(* PLC project HomeAutomation.project, CODESYS CODESYS V3.5 SP15 Patch 1 *)
(* stored: creationDateTime 2019-10-07T17:20:35.7601886, modificationDateTime 2019-10-07T17:17:55.9764537 *)

TYPE MQTT_MESSAGE : STRUCT
  Payload : STRING(128);
  Topic : STRING(128);
  Qos : SD_MQTT.QoS;
  MqttRetain : BOOL;
END_STRUCT;
END_TYPE

TYPE COVER_STATES : (Idle, Auto, Manual, Prio_up, Prio_dn, Calibrate_up, Calibrate_dn);
END_TYPE

PROGRAM PLC_PRG_MAIN
  VAR
    MqttPushbuttonPrefix : STRING(100) := 'WAGO-PFC200/Out/DigitalInputs/Pushbuttons/';  (* INPUT FUNCTION BLOCKS *)
    FB_DI_PB_001 : FB_INPUT_PUSHBUTTON_MQTT;
    FB_DI_PB_002 : FB_INPUT_PUSHBUTTON_MQTT;
    FB_DI_PB_003 : FB_INPUT_PUSHBUTTON_MQTT;
    FB_DI_PB_004 : FB_INPUT_PUSHBUTTON_MQTT;
    FB_DI_PB_005 : FB_INPUT_PUSHBUTTON_MQTT;
    FB_DI_PB_006 : FB_INPUT_PUSHBUTTON_MQTT;
    FB_DI_PB_007 : FB_INPUT_PUSHBUTTON_MQTT;
    FB_DI_PB_008 : FB_INPUT_PUSHBUTTON_MQTT;
    FB_DI_PB_009 : FB_INPUT_PUSHBUTTON_DIMMER_MQTT;
    FB_DI_PB_010 : FB_INPUT_PUSHBUTTON_MQTT;
    FB_DI_PB_011 : FB_INPUT_PUSHBUTTON_MQTT;
    FB_DI_PB_012 : FB_INPUT_PUSHBUTTON_MQTT;
    FB_DI_PB_013 : FB_INPUT_PUSHBUTTON_MQTT;
    FB_DI_PB_014 : FB_INPUT_PUSHBUTTON_MQTT;
    FB_DI_PB_015 : FB_INPUT_PUSHBUTTON_MQTT;
    FB_DI_PB_016 : FB_INPUT_PUSHBUTTON_MQTT;
    FB_DI_PB_017 : FB_INPUT_PUSHBUTTON_MQTT;
    FB_DI_PB_018 : FB_INPUT_PUSHBUTTON_MQTT;
    FB_DI_PB_019 : FB_INPUT_PUSHBUTTON_MQTT;
    FB_DI_PB_020 : FB_INPUT_PUSHBUTTON_MQTT;
    FB_DI_PB_021 : FB_INPUT_PUSHBUTTON_MQTT;
    FB_DI_PB_022 : FB_INPUT_PUSHBUTTON_MQTT;
    FB_DI_PB_023 : FB_INPUT_PUSHBUTTON_MQTT;
    FB_DI_PB_024 : FB_INPUT_PUSHBUTTON_MQTT;
    FB_DI_PB_025 : FB_INPUT_PUSHBUTTON_MQTT;
    FB_DI_PB_026 : FB_INPUT_PUSHBUTTON_MQTT;
    FB_DI_PB_027 : FB_INPUT_PUSHBUTTON_MQTT;
    FB_DI_PB_028 : FB_INPUT_PUSHBUTTON_MQTT;
    FB_DI_PB_029 : FB_INPUT_PUSHBUTTON_MQTT;
    FB_DI_PB_030 : FB_INPUT_PUSHBUTTON_MQTT;
    FB_DI_PB_031 : FB_INPUT_PUSHBUTTON_MQTT;
    FB_DI_PB_032 : FB_INPUT_PUSHBUTTON_MQTT;
    FB_DI_PB_033 : FB_INPUT_PUSHBUTTON_MQTT;
    FB_DI_PB_034 : FB_INPUT_PUSHBUTTON_MQTT;
    FB_DI_PB_035 : FB_INPUT_PUSHBUTTON_MQTT;
    FB_DI_PB_036 : FB_INPUT_PUSHBUTTON_MQTT;
    FB_DI_PB_037 : FB_INPUT_PUSHBUTTON_MQTT;
    FB_DI_PB_038 : FB_INPUT_PUSHBUTTON_MQTT;
    FB_DI_PB_039 : FB_INPUT_PUSHBUTTON_MQTT;
    FB_DI_PB_040 : FB_INPUT_PUSHBUTTON_MQTT;
    FB_DI_PB_041 : FB_INPUT_PUSHBUTTON_MQTT;
    FB_DI_PB_042 : FB_INPUT_PUSHBUTTON_MQTT;
    FB_DI_PB_043 : FB_INPUT_PUSHBUTTON_MQTT;
    FB_DI_PB_044 : FB_INPUT_PUSHBUTTON_MQTT;
    FB_DI_PB_045 : FB_INPUT_PUSHBUTTON_MQTT;
    FB_DI_PB_046 : FB_INPUT_PUSHBUTTON_MQTT;
    FB_DI_PB_047 : FB_INPUT_PUSHBUTTON_MQTT;
    FB_DI_PB_048 : FB_INPUT_PUSHBUTTON_MQTT;
    MqttPubSwitchPrefix : STRING(100) := 'WAGO-PFC200/Out/DigitalOutputs/';  (* OUTPUT FUNCTION BLOCKS *)
    MqttSubSwitchPrefix : STRING(100) := 'WAGO-PFC200/In/DigitalOutputs/';
    FB_DO_SW_001 : FB_OUTPUT_SWITCH_MQTT;
    FB_DO_SW_002 : FB_OUTPUT_SWITCH_MQTT;
    FB_DO_SW_003 : FB_OUTPUT_SWITCH_MQTT;
    FB_DO_SW_004 : FB_OUTPUT_SWITCH_MQTT;
    FB_DO_SW_005 : FB_OUTPUT_SWITCH_MQTT;
    FB_DO_SW_006 : FB_OUTPUT_SWITCH_MQTT;
    FB_DO_SW_007 : FB_OUTPUT_SWITCH_MQTT;
    FB_DO_SW_008 : FB_OUTPUT_SWITCH_MQTT;
    FB_DO_SW_009 : FB_OUTPUT_SWITCH_MQTT;
    FB_DO_SW_010 : FB_OUTPUT_SWITCH_MQTT;
    FB_DO_SW_011 : FB_OUTPUT_SWITCH_MQTT;
    FB_DO_SW_012 : FB_OUTPUT_SWITCH_MQTT;
    FB_DO_SW_013 : FB_OUTPUT_SWITCH_MQTT;
    FB_DO_SW_014 : FB_OUTPUT_SWITCH_MQTT;
    FB_DO_SW_015 : FB_OUTPUT_SWITCH_MQTT;
    FB_DO_SW_016 : FB_OUTPUT_SWITCH_MQTT;
    FB_DO_SW_017 : FB_OUTPUT_SWITCH_MQTT;
    FB_DO_SW_018 : FB_OUTPUT_SWITCH_MQTT;
    FB_DO_SW_019 : FB_OUTPUT_SWITCH_MQTT;
    FB_DO_SW_020 : FB_OUTPUT_SWITCH_MQTT;
    FB_DO_SW_021 : FB_OUTPUT_SWITCH_MQTT;
    FB_DO_SW_022 : FB_OUTPUT_SWITCH_MQTT;
    FB_DO_SW_023 : FB_OUTPUT_SWITCH_MQTT;
    FB_DO_SW_024 : FB_OUTPUT_SWITCH_MQTT;
    FB_DO_SW_025 : FB_OUTPUT_SWITCH_MQTT;
    FB_DO_SW_026 : FB_OUTPUT_SWITCH_MQTT;
    FB_DO_SW_027 : FB_OUTPUT_SWITCH_MQTT;
    FB_DO_SW_028 : FB_OUTPUT_SWITCH_MQTT;
    FB_DO_SW_029 : FB_OUTPUT_SWITCH_MQTT;
    FB_DO_SW_030 : FB_OUTPUT_SWITCH_MQTT;
    FB_DO_SW_031 : FB_OUTPUT_SWITCH_MQTT;
    FB_DO_SW_032 : FB_OUTPUT_SWITCH_MQTT;
    MqttPubCoverPrefix : STRING(100) := 'WAGO-PFC200/Out/Covers/';  (* COVER FUNCTION BLOCKS *)
    MqttSubCoverPrefix : STRING(100) := 'WAGO-PFC200/In/Covers/';
    FB_DO_COVER_001 : FB_OUTPUT_COVER_MQTT;
  END_VAR

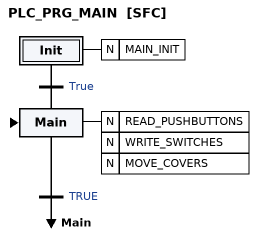
INITIAL_STEP Init:
  MAIN_INIT(N);
END_STEP
TRANSITION FROM Init TO Main
  := True;
END_TRANSITION
STEP Main:
  READ_PUSHBUTTONS(N);
  WRITE_SWITCHES(N);
  MOVE_COVERS(N);
END_STEP
TRANSITION FROM Main TO Main
  := TRUE;
END_TRANSITION

ACTION WRITE_SWITCHES:
                      FB_DO_SW_001(OUT	=>		DO_001,										(* couple the function block to the physical output *)
	PRIO_HIGH				:=FALSE,  									(* brings the output high regardless of other input values *)
	PRIO_LOW				:=FALSE, 									(* brings the output low regardless of other input values. NOTE: PRIO_HIGH overrules PRIO_LOW input *)
	TOGGLE					:=FB_DI_PB_009.SINGLE 						(* for toggling the output *)	
);

FB_DO_SW_002(OUT => DO_002		,PRIO_HIGH:=FALSE			,PRIO_LOW:=FALSE				,TOGGLE:=FB_DI_PB_009.DOUBLE	);
FB_DO_SW_003(OUT => DO_003		,PRIO_HIGH:=FALSE			,PRIO_LOW:=FALSE				,TOGGLE:=FB_DI_PB_009.LONG		);
FB_DO_SW_004(OUT => DO_004		,PRIO_HIGH:=FALSE			,PRIO_LOW:=FALSE				,TOGGLE:=FB_DI_PB_009.LONG		);
FB_DO_SW_005(OUT => DO_005		,PRIO_HIGH:=FALSE			,PRIO_LOW:=FALSE				,TOGGLE:=FB_DI_PB_009.LONG		);
FB_DO_SW_006(OUT => DO_006		,PRIO_HIGH:=FALSE			,PRIO_LOW:=FALSE				,TOGGLE:=FB_DI_PB_009.LONG		);
FB_DO_SW_007(OUT => DO_007		,PRIO_HIGH:=FALSE			,PRIO_LOW:=FALSE				,TOGGLE:=FB_DI_PB_009.LONG		);
FB_DO_SW_008(OUT => DO_008		,PRIO_HIGH:=FALSE			,PRIO_LOW:=FALSE				,TOGGLE:=FB_DI_PB_009.LONG		);
FB_DO_SW_009(OUT => DO_009		,PRIO_HIGH:=FALSE			,PRIO_LOW:=FALSE				,TOGGLE:=FALSE				);
FB_DO_SW_010(OUT => DO_010		,PRIO_HIGH:=FALSE			,PRIO_LOW:=FALSE				,TOGGLE:=FALSE				);
FB_DO_SW_011(OUT => DO_011		,PRIO_HIGH:=FALSE			,PRIO_LOW:=FALSE				,TOGGLE:=FALSE				);
FB_DO_SW_012(OUT => DO_012		,PRIO_HIGH:=FALSE			,PRIO_LOW:=FALSE				,TOGGLE:=FALSE				);
FB_DO_SW_013(OUT => DO_013		,PRIO_HIGH:=FALSE			,PRIO_LOW:=FALSE				,TOGGLE:=FALSE				);
FB_DO_SW_014(OUT => DO_014		,PRIO_HIGH:=FALSE			,PRIO_LOW:=FALSE				,TOGGLE:=FALSE				);
FB_DO_SW_015(OUT => DO_015		,PRIO_HIGH:=FALSE			,PRIO_LOW:=FALSE				,TOGGLE:=FALSE				);
FB_DO_SW_016(OUT => DO_016		,PRIO_HIGH:=FALSE			,PRIO_LOW:=FALSE				,TOGGLE:=FALSE				);
FB_DO_SW_017(OUT => DO_017		,PRIO_HIGH:=FALSE			,PRIO_LOW:=FALSE				,TOGGLE:=FALSE				);
FB_DO_SW_018(OUT => DO_018		,PRIO_HIGH:=FALSE			,PRIO_LOW:=FALSE				,TOGGLE:=FALSE				);
FB_DO_SW_019(OUT => DO_019		,PRIO_HIGH:=FALSE			,PRIO_LOW:=FALSE				,TOGGLE:=FALSE				);
FB_DO_SW_020(OUT => DO_020		,PRIO_HIGH:=FALSE			,PRIO_LOW:=FALSE				,TOGGLE:=FALSE				);
FB_DO_SW_021(OUT => DO_021		,PRIO_HIGH:=FALSE			,PRIO_LOW:=FALSE				,TOGGLE:=FALSE				);
FB_DO_SW_022(OUT => DO_022		,PRIO_HIGH:=FALSE			,PRIO_LOW:=FALSE				,TOGGLE:=FALSE				);
FB_DO_SW_023(OUT => DO_023		,PRIO_HIGH:=FALSE			,PRIO_LOW:=FALSE				,TOGGLE:=FALSE				);
FB_DO_SW_024(OUT => DO_024		,PRIO_HIGH:=FALSE			,PRIO_LOW:=FALSE				,TOGGLE:=FALSE				);
FB_DO_SW_025(OUT => DO_025		,PRIO_HIGH:=FALSE			,PRIO_LOW:=FALSE				,TOGGLE:=FALSE				);
FB_DO_SW_026(OUT => DO_026		,PRIO_HIGH:=FALSE			,PRIO_LOW:=FALSE				,TOGGLE:=FALSE				);
FB_DO_SW_027(OUT => DO_027		,PRIO_HIGH:=FALSE			,PRIO_LOW:=FALSE				,TOGGLE:=FALSE				);
FB_DO_SW_028(OUT => DO_028		,PRIO_HIGH:=FALSE			,PRIO_LOW:=FALSE				,TOGGLE:=FALSE				);
FB_DO_SW_029(OUT => DO_029		,PRIO_HIGH:=FALSE			,PRIO_LOW:=FALSE				,TOGGLE:=FALSE				);
FB_DO_SW_030(OUT => DO_030		,PRIO_HIGH:=FALSE			,PRIO_LOW:=FALSE				,TOGGLE:=FALSE				);

                    
END_ACTION

ACTION READ_PUSHBUTTONS:
                      FB_DI_PB_001(PB:= DI_001); (* Provide the input FB the correct phyical input to validate each cyclus *)
FB_DI_PB_002(PB:= DI_002);
FB_DI_PB_003(PB:= DI_003);
FB_DI_PB_004(PB:= DI_004);
FB_DI_PB_005(PB:= DI_005);
FB_DI_PB_006(PB:= DI_006);
FB_DI_PB_007(PB:= DI_007);
FB_DI_PB_008(PB:= DI_008);
FB_DI_PB_009(PB:= DI_009);
FB_DI_PB_010(PB:= DI_010);
FB_DI_PB_011(PB:= DI_011);
FB_DI_PB_012(PB:= DI_012);
FB_DI_PB_013(PB:= DI_013);
FB_DI_PB_014(PB:= DI_014);
FB_DI_PB_015(PB:= DI_015);
FB_DI_PB_016(PB:= DI_016);
FB_DI_PB_017(PB:= DI_017);
FB_DI_PB_018(PB:= DI_018);
FB_DI_PB_019(PB:= DI_019);
FB_DI_PB_020(PB:= DI_020);
FB_DI_PB_021(PB:= DI_021);
FB_DI_PB_022(PB:= DI_022);
FB_DI_PB_023(PB:= DI_023);
FB_DI_PB_024(PB:= DI_024);
FB_DI_PB_025(PB:= DI_025);
FB_DI_PB_026(PB:= DI_026);
FB_DI_PB_027(PB:= DI_027);
FB_DI_PB_028(PB:= DI_028);
FB_DI_PB_029(PB:= DI_029);
FB_DI_PB_030(PB:= DI_030);
FB_DI_PB_031(PB:= DI_031);
FB_DI_PB_032(PB:= DI_032);
FB_DI_PB_033(PB:= DI_033);
FB_DI_PB_034(PB:= DI_034);
FB_DI_PB_035(PB:= DI_035);
FB_DI_PB_036(PB:= DI_036);
FB_DI_PB_037(PB:= DI_037);
FB_DI_PB_038(PB:= DI_038);
FB_DI_PB_039(PB:= DI_039);
FB_DI_PB_040(PB:= DI_040);
FB_DI_PB_041(PB:= DI_041);
FB_DI_PB_042(PB:= DI_042);
FB_DI_PB_043(PB:= DI_043);
FB_DI_PB_044(PB:= DI_044);
FB_DI_PB_045(PB:= DI_045);
FB_DI_PB_046(PB:= DI_046);
FB_DI_PB_047(PB:= DI_047);
FB_DI_PB_048(PB:= DI_048);
                    
END_ACTION

ACTION MAIN_INIT:
                      (* INIT DIGITAL INPUT STUFF *)
FB_DI_PB_001.InitMqtt(MQTTPublishPrefix:= ADR(MqttPushbuttonPrefix),	(* pointer to string prefix for the mqtt publish topic *)
	pMqttPublishQueue := ADR(MqttVariables.fbMqttPublishQueue)		(* pointer to MqttPublishQueue to send a new Mqtt event *)
);
FB_DI_PB_002.InitMqtt(MQTTPublishPrefix:= ADR(MqttPushbuttonPrefix),	pMqttPublishQueue := ADR(MqttVariables.fbMqttPublishQueue));
FB_DI_PB_003.InitMqtt(MQTTPublishPrefix:= ADR(MqttPushbuttonPrefix),	pMqttPublishQueue := ADR(MqttVariables.fbMqttPublishQueue));
FB_DI_PB_004.InitMqtt(MQTTPublishPrefix:= ADR(MqttPushbuttonPrefix),	pMqttPublishQueue := ADR(MqttVariables.fbMqttPublishQueue));
FB_DI_PB_005.InitMqtt(MQTTPublishPrefix:= ADR(MqttPushbuttonPrefix),	pMqttPublishQueue := ADR(MqttVariables.fbMqttPublishQueue));
FB_DI_PB_006.InitMqtt(MQTTPublishPrefix:= ADR(MqttPushbuttonPrefix),	pMqttPublishQueue := ADR(MqttVariables.fbMqttPublishQueue));
FB_DI_PB_007.InitMqtt(MQTTPublishPrefix:= ADR(MqttPushbuttonPrefix),	pMqttPublishQueue := ADR(MqttVariables.fbMqttPublishQueue));
FB_DI_PB_008.InitMqtt(MQTTPublishPrefix:= ADR(MqttPushbuttonPrefix),	pMqttPublishQueue := ADR(MqttVariables.fbMqttPublishQueue));
FB_DI_PB_009.InitMqtt(MQTTPublishPrefix:= ADR(MqttPushbuttonPrefix),	pMqttPublishQueue := ADR(MqttVariables.fbMqttPublishQueue), TRUE, SD_MQTT.QoS.ExactlyOnce, 5);
FB_DI_PB_010.InitMqtt(MQTTPublishPrefix:= ADR(MqttPushbuttonPrefix),	pMqttPublishQueue := ADR(MqttVariables.fbMqttPublishQueue));
FB_DI_PB_011.InitMqtt(MQTTPublishPrefix:= ADR(MqttPushbuttonPrefix),	pMqttPublishQueue := ADR(MqttVariables.fbMqttPublishQueue));
FB_DI_PB_012.InitMqtt(MQTTPublishPrefix:= ADR(MqttPushbuttonPrefix),	pMqttPublishQueue := ADR(MqttVariables.fbMqttPublishQueue));
FB_DI_PB_013.InitMqtt(MQTTPublishPrefix:= ADR(MqttPushbuttonPrefix),	pMqttPublishQueue := ADR(MqttVariables.fbMqttPublishQueue));
FB_DI_PB_014.InitMqtt(MQTTPublishPrefix:= ADR(MqttPushbuttonPrefix),	pMqttPublishQueue := ADR(MqttVariables.fbMqttPublishQueue));
FB_DI_PB_015.InitMqtt(MQTTPublishPrefix:= ADR(MqttPushbuttonPrefix),	pMqttPublishQueue := ADR(MqttVariables.fbMqttPublishQueue));
FB_DI_PB_016.InitMqtt(MQTTPublishPrefix:= ADR(MqttPushbuttonPrefix),	pMqttPublishQueue := ADR(MqttVariables.fbMqttPublishQueue));

(* INIT DIGITAL OUTPUT STUFF *)
FB_DO_SW_001.InitMqtt(MQTTPublishPrefix:= ADR(MqttPubSwitchPrefix),					(* pointer to string prefix for the mqtt publish topic *)
	MQTTSubscribePrefix:= ADR(MqttSubSwitchPrefix),									(* pointer to string prefix for the mqtt subscribe topic *)
	pMqttPublishQueue := ADR(MqttVariables.fbMqttPublishQueue),						(* pointer to MqttPublishQueue to send a new Mqtt event *)
	pMqttCallbackCollector := ADR(MqttVariables.collector_FB_OUTPUT_SWITCH_MQTT)	(* pointer to CallbackCollector to receive Mqtt subscription events *)
);
FB_DO_SW_002.InitMqtt(MQTTPublishPrefix:= ADR(MqttPubSwitchPrefix),	MQTTSubscribePrefix:= ADR(MqttSubSwitchPrefix), pMqttPublishQueue := ADR(MqttVariables.fbMqttPublishQueue), pMqttCallbackCollector := ADR(MqttVariables.collector_FB_OUTPUT_SWITCH_MQTT));
FB_DO_SW_003.InitMqtt(MQTTPublishPrefix:= ADR(MqttPubSwitchPrefix),	MQTTSubscribePrefix:= ADR(MqttSubSwitchPrefix),	pMqttPublishQueue := ADR(MqttVariables.fbMqttPublishQueue), pMqttCallbackCollector := ADR(MqttVariables.collector_FB_OUTPUT_SWITCH_MQTT));
FB_DO_SW_004.InitMqtt(MQTTPublishPrefix:= ADR(MqttPubSwitchPrefix),	MQTTSubscribePrefix:= ADR(MqttSubSwitchPrefix),	pMqttPublishQueue := ADR(MqttVariables.fbMqttPublishQueue), pMqttCallbackCollector := ADR(MqttVariables.collector_FB_OUTPUT_SWITCH_MQTT));
FB_DO_SW_005.InitMqtt(MQTTPublishPrefix:= ADR(MqttPubSwitchPrefix),	MQTTSubscribePrefix:= ADR(MqttSubSwitchPrefix),	pMqttPublishQueue := ADR(MqttVariables.fbMqttPublishQueue), pMqttCallbackCollector := ADR(MqttVariables.collector_FB_OUTPUT_SWITCH_MQTT));
FB_DO_SW_006.InitMqtt(MQTTPublishPrefix:= ADR(MqttPubSwitchPrefix),	MQTTSubscribePrefix:= ADR(MqttSubSwitchPrefix),	pMqttPublishQueue := ADR(MqttVariables.fbMqttPublishQueue), pMqttCallbackCollector := ADR(MqttVariables.collector_FB_OUTPUT_SWITCH_MQTT));
FB_DO_SW_007.InitMqtt(MQTTPublishPrefix:= ADR(MqttPubSwitchPrefix),	MQTTSubscribePrefix:= ADR(MqttSubSwitchPrefix),	pMqttPublishQueue := ADR(MqttVariables.fbMqttPublishQueue), pMqttCallbackCollector := ADR(MqttVariables.collector_FB_OUTPUT_SWITCH_MQTT));
FB_DO_SW_008.InitMqtt(MQTTPublishPrefix:= ADR(MqttPubSwitchPrefix),	MQTTSubscribePrefix:= ADR(MqttSubSwitchPrefix),	pMqttPublishQueue := ADR(MqttVariables.fbMqttPublishQueue), pMqttCallbackCollector := ADR(MqttVariables.collector_FB_OUTPUT_SWITCH_MQTT));
FB_DO_SW_009.InitMqtt(MQTTPublishPrefix:= ADR(MqttPubSwitchPrefix),	MQTTSubscribePrefix:= ADR(MqttSubSwitchPrefix),	pMqttPublishQueue := ADR(MqttVariables.fbMqttPublishQueue), pMqttCallbackCollector := ADR(MqttVariables.collector_FB_OUTPUT_SWITCH_MQTT));
FB_DO_SW_010.InitMqtt(MQTTPublishPrefix:= ADR(MqttPubSwitchPrefix),	MQTTSubscribePrefix:= ADR(MqttSubSwitchPrefix),	pMqttPublishQueue := ADR(MqttVariables.fbMqttPublishQueue), pMqttCallbackCollector := ADR(MqttVariables.collector_FB_OUTPUT_SWITCH_MQTT));
FB_DO_SW_011.InitMqtt(MQTTPublishPrefix:= ADR(MqttPubSwitchPrefix),	MQTTSubscribePrefix:= ADR(MqttSubSwitchPrefix),	pMqttPublishQueue := ADR(MqttVariables.fbMqttPublishQueue), pMqttCallbackCollector := ADR(MqttVariables.collector_FB_OUTPUT_SWITCH_MQTT));
FB_DO_SW_012.InitMqtt(MQTTPublishPrefix:= ADR(MqttPubSwitchPrefix),	MQTTSubscribePrefix:= ADR(MqttSubSwitchPrefix), pMqttPublishQueue := ADR(MqttVariables.fbMqttPublishQueue), pMqttCallbackCollector := ADR(MqttVariables.collector_FB_OUTPUT_SWITCH_MQTT));
FB_DO_SW_013.InitMqtt(MQTTPublishPrefix:= ADR(MqttPubSwitchPrefix),	MQTTSubscribePrefix:= ADR(MqttSubSwitchPrefix), pMqttPublishQueue := ADR(MqttVariables.fbMqttPublishQueue), pMqttCallbackCollector := ADR(MqttVariables.collector_FB_OUTPUT_SWITCH_MQTT));
FB_DO_SW_014.InitMqtt(MQTTPublishPrefix:= ADR(MqttPubSwitchPrefix),	MQTTSubscribePrefix:= ADR(MqttSubSwitchPrefix), pMqttPublishQueue := ADR(MqttVariables.fbMqttPublishQueue), pMqttCallbackCollector := ADR(MqttVariables.collector_FB_OUTPUT_SWITCH_MQTT));
FB_DO_SW_015.InitMqtt(MQTTPublishPrefix:= ADR(MqttPubSwitchPrefix),	MQTTSubscribePrefix:= ADR(MqttSubSwitchPrefix), pMqttPublishQueue := ADR(MqttVariables.fbMqttPublishQueue), pMqttCallbackCollector := ADR(MqttVariables.collector_FB_OUTPUT_SWITCH_MQTT));
FB_DO_SW_016.InitMqtt(MQTTPublishPrefix:= ADR(MqttPubSwitchPrefix),	MQTTSubscribePrefix:= ADR(MqttSubSwitchPrefix), pMqttPublishQueue := ADR(MqttVariables.fbMqttPublishQueue), pMqttCallbackCollector := ADR(MqttVariables.collector_FB_OUTPUT_SWITCH_MQTT));
FB_DO_SW_017.InitMqtt(MQTTPublishPrefix:= ADR(MqttPubSwitchPrefix),	MQTTSubscribePrefix:= ADR(MqttSubSwitchPrefix), pMqttPublishQueue := ADR(MqttVariables.fbMqttPublishQueue), pMqttCallbackCollector := ADR(MqttVariables.collector_FB_OUTPUT_SWITCH_MQTT));
FB_DO_SW_018.InitMqtt(MQTTPublishPrefix:= ADR(MqttPubSwitchPrefix),	MQTTSubscribePrefix:= ADR(MqttSubSwitchPrefix), pMqttPublishQueue := ADR(MqttVariables.fbMqttPublishQueue), pMqttCallbackCollector := ADR(MqttVariables.collector_FB_OUTPUT_SWITCH_MQTT));
FB_DO_SW_019.InitMqtt(MQTTPublishPrefix:= ADR(MqttPubSwitchPrefix),	MQTTSubscribePrefix:= ADR(MqttSubSwitchPrefix), pMqttPublishQueue := ADR(MqttVariables.fbMqttPublishQueue), pMqttCallbackCollector := ADR(MqttVariables.collector_FB_OUTPUT_SWITCH_MQTT));
FB_DO_SW_020.InitMqtt(MQTTPublishPrefix:= ADR(MqttPubSwitchPrefix),	MQTTSubscribePrefix:= ADR(MqttSubSwitchPrefix), pMqttPublishQueue := ADR(MqttVariables.fbMqttPublishQueue), pMqttCallbackCollector := ADR(MqttVariables.collector_FB_OUTPUT_SWITCH_MQTT));
FB_DO_SW_021.InitMqtt(MQTTPublishPrefix:= ADR(MqttPubSwitchPrefix),	MQTTSubscribePrefix:= ADR(MqttSubSwitchPrefix), pMqttPublishQueue := ADR(MqttVariables.fbMqttPublishQueue), pMqttCallbackCollector := ADR(MqttVariables.collector_FB_OUTPUT_SWITCH_MQTT));
FB_DO_SW_022.InitMqtt(MQTTPublishPrefix:= ADR(MqttPubSwitchPrefix),	MQTTSubscribePrefix:= ADR(MqttSubSwitchPrefix), pMqttPublishQueue := ADR(MqttVariables.fbMqttPublishQueue), pMqttCallbackCollector := ADR(MqttVariables.collector_FB_OUTPUT_SWITCH_MQTT));
FB_DO_SW_023.InitMqtt(MQTTPublishPrefix:= ADR(MqttPubSwitchPrefix),	MQTTSubscribePrefix:= ADR(MqttSubSwitchPrefix), pMqttPublishQueue := ADR(MqttVariables.fbMqttPublishQueue), pMqttCallbackCollector := ADR(MqttVariables.collector_FB_OUTPUT_SWITCH_MQTT));
FB_DO_SW_024.InitMqtt(MQTTPublishPrefix:= ADR(MqttPubSwitchPrefix),	MQTTSubscribePrefix:= ADR(MqttSubSwitchPrefix), pMqttPublishQueue := ADR(MqttVariables.fbMqttPublishQueue), pMqttCallbackCollector := ADR(MqttVariables.collector_FB_OUTPUT_SWITCH_MQTT));
FB_DO_SW_025.InitMqtt(MQTTPublishPrefix:= ADR(MqttPubSwitchPrefix),	MQTTSubscribePrefix:= ADR(MqttSubSwitchPrefix), pMqttPublishQueue := ADR(MqttVariables.fbMqttPublishQueue), pMqttCallbackCollector := ADR(MqttVariables.collector_FB_OUTPUT_SWITCH_MQTT));
FB_DO_SW_026.InitMqtt(MQTTPublishPrefix:= ADR(MqttPubSwitchPrefix),	MQTTSubscribePrefix:= ADR(MqttSubSwitchPrefix), pMqttPublishQueue := ADR(MqttVariables.fbMqttPublishQueue), pMqttCallbackCollector := ADR(MqttVariables.collector_FB_OUTPUT_SWITCH_MQTT));
FB_DO_SW_027.InitMqtt(MQTTPublishPrefix:= ADR(MqttPubSwitchPrefix),	MQTTSubscribePrefix:= ADR(MqttSubSwitchPrefix), pMqttPublishQueue := ADR(MqttVariables.fbMqttPublishQueue), pMqttCallbackCollector := ADR(MqttVariables.collector_FB_OUTPUT_SWITCH_MQTT));
FB_DO_SW_028.InitMqtt(MQTTPublishPrefix:= ADR(MqttPubSwitchPrefix),	MQTTSubscribePrefix:= ADR(MqttSubSwitchPrefix), pMqttPublishQueue := ADR(MqttVariables.fbMqttPublishQueue), pMqttCallbackCollector := ADR(MqttVariables.collector_FB_OUTPUT_SWITCH_MQTT));
FB_DO_SW_029.InitMqtt(MQTTPublishPrefix:= ADR(MqttPubSwitchPrefix),	MQTTSubscribePrefix:= ADR(MqttSubSwitchPrefix), pMqttPublishQueue := ADR(MqttVariables.fbMqttPublishQueue), pMqttCallbackCollector := ADR(MqttVariables.collector_FB_OUTPUT_SWITCH_MQTT));
FB_DO_SW_030.InitMqtt(MQTTPublishPrefix:= ADR(MqttPubSwitchPrefix),	MQTTSubscribePrefix:= ADR(MqttSubSwitchPrefix), pMqttPublishQueue := ADR(MqttVariables.fbMqttPublishQueue), pMqttCallbackCollector := ADR(MqttVariables.collector_FB_OUTPUT_SWITCH_MQTT));

(* INIT COVERS STUFF *)
FB_DO_COVER_001.InitMqtt(MQTTPublishPrefix:= ADR(MqttPubCoverPrefix),				(* pointer to string prefix for the mqtt publish topic *)
	MQTTSubscribePrefix:= ADR(MqttSubCoverPrefix),									(* pointer to string prefix for the mqtt subscribe topic *)
	pMqttPublishQueue := ADR(MqttVariables.fbMqttPublishQueue),						(* pointer to MqttPublishQueue to send a new Mqtt event *)
	pMqttCallbackCollector := ADR(MqttVariables.collector_FB_OUTPUT_COVER_MQTT), 	(* pointer to CallbackCollector to receive Mqtt subscription events *)
	SD_MQTT.QoS.ExactlyOnce, 														(* specify the QoS for the POS mqtt events (values 0-100) *)
	2																				(* specify the resolution for the POS mqtt events *)
);

FB_DO_COVER_001.ConfigureFunctionBlock(T_LOCKOUT:=T#1S,								(* delay between change of direction *)
	T_UD:=T#20S																		(* run time to move the cover completely up/down *)
);
                    
END_ACTION

ACTION MOVE_COVERS:
                      FB_DO_COVER_001(
	UP:=FB_DI_PB_013.P_LONG,
	DN:=FB_DI_PB_015.P_LONG,
	MU=>DO_031,
	MD=>DO_032	
	);
                    
END_ACTION
END_PROGRAM

{attribute 'reflection'}
FUNCTION_BLOCK FB_INPUT_PUSHBUTTON_MQTT
  VAR_INPUT
    PB : BOOL;
  END_VAR
  VAR_OUTPUT
    SINGLE : BOOL;
    DOUBLE : BOOL;
    LONG : BOOL;
    P_LONG : BOOL;
  END_VAR
  VAR
    {attribute 'instance-path'}
    {attribute 'noinit'}
    InstanceName : STRING;  (* object's full instance name *)
    InitMqttDone : BOOL;
    MqttPublishTopicPrefix : POINTER TO STRING;
    MqttPublishTopicSuffix : STRING(15);
    pMqttPublishQueue : POINTER TO FB_MqttPublishQueue;
    FB_DETECTPUSH : OSCAT_BUILDING.CLICK_MODE;
    P_LONG_R_TRIG : Standard.R_TRIG;
    P_LONG_F_TRIG : Standard.F_TRIG;
    T_Long : TIME := TIME#400ms;  (* Default value for click mode, can be overwritten by method call *)
  END_VAR

                  FB_DETECTPUSH(
	IN:= PB, 	
	SINGLE=> SINGLE, 
	DOUBLE=> DOUBLE, 
	TP_LONG=> LONG, 
	LONG=> P_LONG,
	T_LONG:= T_Long);
	
P_LONG_R_TRIG(CLK:=FB_DETECTPUSH.LONG);
P_LONG_F_TRIG(CLK:=FB_DETECTPUSH.LONG);
	
IF FB_DETECTPUSH.SINGLE AND InitMqttDone THEN
	pMqttPublishQueue^.AddMessage(
		Payload := 'SINGLE',
		Topic := CONCAT(MqttPublishTopicPrefix^, MqttPublishTopicSuffix),
		Qos := SD_MQTT.QoS.ExactlyOnce,
		MqttRetain := FALSE
	);
END_IF

IF FB_DETECTPUSH.DOUBLE AND InitMqttDone THEN
	pMqttPublishQueue^.AddMessage(
		Payload := 'DOUBLE',
		Topic := CONCAT(MqttPublishTopicPrefix^, MqttPublishTopicSuffix),
		Qos := SD_MQTT.QoS.ExactlyOnce,
		MqttRetain := FALSE
	);
END_IF

IF FB_DETECTPUSH.TP_LONG AND InitMqttDone THEN
	pMqttPublishQueue^.AddMessage(
		Payload := 'LONG',
		Topic := CONCAT(MqttPublishTopicPrefix^, MqttPublishTopicSuffix),
		Qos := SD_MQTT.QoS.ExactlyOnce,
		MqttRetain := FALSE
	);
END_IF

IF (P_LONG_R_TRIG.Q OR P_LONG_F_TRIG.Q) AND InitMqttDone THEN
	pMqttPublishQueue^.AddMessage(
		Payload := BOOL_TO_STRING(FB_DETECTPUSH.LONG),
		Topic := CONCAT(CONCAT(MqttPublishTopicPrefix^, MqttPublishTopicSuffix),'/P_LONG'),
		Qos := SD_MQTT.QoS.ExactlyOnce,
		MqttRetain := TRUE
	);
END_IF
                

METHOD InitMqtt
  VAR_INPUT
    MQTTPublishPrefix : POINTER TO STRING;
    pMqttPublishQueue : POINTER TO FB_MqttPublishQueue;
  END_VAR
  VAR
    InstanceNamePt : POINTER TO STRING;
  END_VAR
                        THIS^.pMqttPublishQueue := pMqttPublishQueue;
THIS^.MqttPublishTopicPrefix := MQTTPublishPrefix;

InstanceNamePt := CommonTypesAndFunctions.FindLastDot(ADR(THIS^.InstanceName)) + 1;
THIS^.MqttPublishTopicSuffix := InstanceNamePt^;

InitMqttDone := TRUE;
                      
END_METHOD

METHOD ConfigureFunctionBlock
  VAR_INPUT
    T_Long : TIME;  (* Default value for click mode, can be overwritten by method call *)
  END_VAR
                        THIS^.T_Long:=T_Long;
                      
END_METHOD
END_FUNCTION_BLOCK

{attribute 'reflection'}
FUNCTION_BLOCK FB_OUTPUT_SWITCH_MQTT IMPLEMENTS SD_MQTT.MQTT_SUBSCRIBE_CALLBACK
  VAR_INPUT
    PRIO_HIGH : BOOL := FALSE;
    PRIO_LOW : BOOL := FALSE;
    TOGGLE : BOOL := FALSE;
  END_VAR
  VAR_OUTPUT
    OUT : BOOL;
  END_VAR
  VAR
    {attribute 'instance-path'}
    {attribute 'noinit'}
    InstanceName : STRING;  (* object's full instance name *)
    Startup : BOOL := TRUE;
    InitMqttDone : BOOL;
    MqttPublishTopicPrefix : POINTER TO STRING;
    MqttPublishTopicSuffix : STRING(15);
    MQTTSubscribeTopic : STRING(50);
    pMqttPublishQueue : POINTER TO FB_MqttPublishQueue;
    MqttHighRequest : BOOL;
    MqttLowRequest : BOOL;
  END_VAR
  VAR PERSISTENT
    PreviousState : BOOL;  (* To retain output state through powercycles *)
  END_VAR

                  IF Startup THEN
	OUT := PreviousState;
END_IF

IF PRIO_HIGH THEN
	OUT:=TRUE;
ELSIF(PRIO_LOW AND NOT (PRIO_HIGH)) THEN
	OUT:= FALSE;
ELSIF MqttHighRequest THEN
	OUT:= TRUE;
	MqttHighRequest := FALSE;
	MqttLowRequest := FALSE;
ELSIF MqttLowRequest THEN
	OUT:= FALSE;
	MqttHighRequest := FALSE;
	MqttLowRequest := FALSE;
ELSIF(TOGGLE) THEN
	OUT:=NOT(OUT);
END_IF;

IF(PreviousState <> OUT) OR Startup AND InitMqttDone THEN
	pMqttPublishQueue^.AddMessage(
		Payload := BOOL_TO_STRING(OUT),
		Topic := CONCAT(MqttPublishTopicPrefix^, MqttPublishTopicSuffix),
		Qos := SD_MQTT.QoS.ExactlyOnce,
		MqttRetain := TRUE
	);	
	Startup:=FALSE;
END_IF	

PreviousState := OUT;
                

METHOD InitMqtt
  VAR_INPUT
    MQTTPublishPrefix : POINTER TO STRING;
    MQTTSubscribePrefix : POINTER TO STRING;
    pMqttPublishQueue : POINTER TO FB_MqttPublishQueue;
    pMqttCallbackCollector : POINTER TO SD_MQTT.CallbackCollector;
  END_VAR
  VAR
    InstanceNamePt : POINTER TO STRING;
  END_VAR
                        THIS^.pMqttPublishQueue := pMqttPublishQueue;
THIS^.MqttPublishTopicPrefix := MQTTPublishPrefix;

InstanceNamePt := CommonTypesAndFunctions.FindLastDot(ADR(THIS^.InstanceName)) + 1;
THIS^.MqttPublishTopicSuffix := InstanceNamePt^;
THIS^.MQTTSubscribeTopic := CONCAT(MQTTSubscribePrefix^ ,THIS^.MqttPublishTopicSuffix);

// register the FB agains the collector so mqtt events can be received
pMqttCallbackCollector^.put(instance:= THIS^);

InitMqttDone := TRUE;
                      
END_METHOD

METHOD PublishReceived : BOOL
  VAR_INPUT
    Data : SD_MQTT.CALLBACK_DATA;  (* Collection of recived Data *)
  END_VAR
                        //first check if Mqtt is initialized, otherwise do nothing
IF NOT(InitMqttDone) THEN
	//mark the interface call from the collector as done
	PublishReceived := TRUE;
//check if the packet is for this FB
ELSIF CommonTypesAndFunctions.StrEquals(str1:= ADR(MQTTSubscribeTopic), str2:= Data.TopicOut) THEN
	//mark the interface call from the collector as done
	PublishReceived := TRUE;
	//now process the data
	IF CommonTypesAndFunctions.StrEquals(str1:= Data.PayloadString, str2:= ADR('TRUE')) THEN
		MqttHighRequest := TRUE;
	END_IF
	IF CommonTypesAndFunctions.StrEquals(str1:= Data.PayloadString, str2:= ADR('FALSE')) THEN
		MqttLowRequest := TRUE;
	END_IF
END_IF 
                      
END_METHOD
END_FUNCTION_BLOCK

FUNCTION_BLOCK FB_MqttPublishWorker
  VAR_OUTPUT
    SendDone : BOOL;
  END_VAR
  VAR
    LocalMqttMessage : MQTT_MESSAGE;
    InitDone : BOOL;
    RequestToSend : BOOL;
    Send : BOOL;
    publish : SD_MQTT.MQTTPublish;
  END_VAR

                  //need to call publish here because of FB nums
publish(
	Topic:= ADR(LocalMqttMessage.Topic), 
	PayloadString:= ADR(LocalMqttMessage.Payload), 
	PublishAsString:= TRUE, 
	QoSIn:= LocalMqttMessage.Qos, 
	MRetain:= LocalMqttMessage.MqttRetain, 
	send:= Send);
	
IF NOT InitDone THEN RETURN; END_IF

IF RequestToSend THEN
	Send := TRUE;
	SendDone := FALSE;
END_IF

IF publish.done THEN
	 SendDone := TRUE;
	 RequestToSend:=FALSE;
	 Send:=FALSE;
END_IF
                

METHOD Init
  VAR_INPUT
    inputMQTT_IN_OUT : POINTER TO SD_MQTT.MQTT_IN_OUT;  (* Pointer MQTTT exchange strucure *)
  END_VAR
                        publish.SetMqttInOut(MQTT_IN_OUT := inputMQTT_IN_OUT);

InitDone := TRUE;
SendDone := TRUE;

                      
END_METHOD

METHOD PublishMessage
  VAR_INPUT
    MqttMessage : MQTT_MESSAGE;
  END_VAR
                        LocalMqttMessage := MqttMessage;

RequestToSend:=TRUE;
                      
END_METHOD
END_FUNCTION_BLOCK

FUNCTION_BLOCK FB_MqttPublishQueue
  VAR_OUTPUT
    EMPTY : BOOL := TRUE;
    FULL : BOOL;
  END_VAR
  VAR
    localMessage : MQTT_MESSAGE;
    fifo : ARRAY[0..n] OF MQTT_MESSAGE;
    pr : INT;
    pw : INT;
  END_VAR
  VAR CONSTANT
    n : INT := 1024;  (* changing this value will chage the number of stored elements in the fifo *)
  END_VAR

                  
                

METHOD GetMessage : MQTT_MESSAGE
                        IF NOT EMPTY THEN
	GetMessage := fifo[pr];
	pr := OSCAT_BASIC.INC1(pr,n);
	EMPTY := pr = pw;
	FULL := FALSE;
END_IF;
                      
END_METHOD

METHOD AddMessage
  VAR_INPUT
    Payload : STRING(128);
    Topic : STRING(128);
    Qos : SD_MQTT.QoS;
    MqttRetain : BOOL;
  END_VAR
                        IF NOT FULL THEN
	localMessage.Payload := Payload;
	localMessage.Topic := Topic;
	localMessage.Qos := Qos;
	localMessage.MqttRetain := MqttRetain;
	fifo[pw] := localMessage;
	pw := OSCAT_BASIC.INC1(pw,n);
	FULL := pw = pr;
	EMPTY := FALSE;
END_IF;
                      
END_METHOD

METHOD Reset
                        pw := pr;
FULL := FALSE;
EMPTY := TRUE;
                      
END_METHOD
END_FUNCTION_BLOCK

PROGRAM PLC_PRG_MQTT
  VAR
    broker : STRING := '192.168.1.36:1883';  (* variables for MQTT configuration *)
    clientID : STRING := 'WAGO-PFC200';  (* use the below for username password authentication to broker broker :STRING:='user:password@192.168.1.36:1883'; *)
    MQTTClient : SD_MQTT.HANDLE_MQTT;
    MQTT_IN_OUT : SD_MQTT.MQTT_IN_OUT;
    MQTTInfo : SD_MQTT.MQTT_INFO;
    MQTTLwtTopic : STRING := 'Devices/WAGO-PFC200/availability';
    MQTTLwtPayload : STRING := 'offline';
    MQTTBirthMessage : MQTT_MESSAGE;
    MQTTBirthTopic : STRING := 'Devices/WAGO-PFC200/availability';
    MQTTBirthPayload : STRING := 'online';
    MQTTBirthHartbeat : OSCAT_BASIC.GEN_PULSE;
    MQTTBirthHartbeatTime : TIME := TIME#5s0ms;
    MQTTConnectTrigger : Standard.R_TRIG;
    MQTTPublishBirth : BOOL := TRUE;
    MQTTBirthPublisher : FB_MqttPublishWorker;
    initMqtt : BOOL;  (* variables for MQTT setup *)
    icounter : UDINT;
    ipublishers : UDINT := 40;  (* variables for MQTT publishing *)
    publishers : ARRAY[0..39] OF FB_MqttPublishWorker;
    i : UDINT;  (* variables to work with Mqttbuffer *)
    subscriber_FB_OUTPUT_SWITCH_MQTT : SD_MQTT.MQTTSubscribe;  (* variables for MQTT subscribing *)
    subscriber_FB_OUTPUT_COVER_MQTT : SD_MQTT.MQTTSubscribe;
  END_VAR

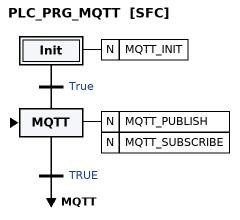
INITIAL_STEP Init:
  MQTT_INIT(N);
END_STEP
TRANSITION FROM Init TO MQTT
  := True;
END_TRANSITION
STEP MQTT:
  MQTT_PUBLISH(N);
  MQTT_SUBSCRIBE(N);
END_STEP
TRANSITION FROM MQTT TO MQTT
  := TRUE;
END_TRANSITION

ACTION MQTT_INIT:
                      
IF NOT initMqtt THEN
	initMqtt := TRUE;
	(* Basic MQTT config *)
	MQTT_IN_OUT.ClientID := clientID;
	
	(* Set the LWT topic / payload *)
	MQTT_IN_OUT.BuildWillTopicAndMessage := FALSE;
	MQTT_IN_OUT.WillTopicBase := '';
	MQTT_IN_OUT.ClientWillTopic := MQTTLwtTopic;
	MQTT_IN_OUT.ClientWillMessage := MQTTLwtPayload;
	
	(* Set the birth message *)
	MQTTBirthMessage.Payload := MQTTBirthPayload;
	MQTTBirthMessage.Topic := MQTTBirthTopic;
	MQTTBirthMessage.Qos := SD_MQTT.QoS.ExactlyOnce;
	MQTTBirthMessage.MqttRetain := FALSE;
	
	(* Configure the rising edge detector to detect a connect/reconnect to the broker, used for  birth message *)
	MQTTConnectTrigger(CLK := MQTTInfo.MQTT_CONNECTED);
	
	(* Configure the dedicated MQTTBirth publisher *)
	MQTTBirthPublisher.Init(inputMQTT_IN_OUT:= ADR(MQTT_IN_OUT));
	
	(* Configure the pulse generator for the birth message hartbeat *)
	 MQTTBirthHartbeat(ENQ:=TRUE, PTH:=T#0S, PTL:=MQTTBirthHartbeatTime);
	
	(* INIT MQTT PUBLISH STUFF *)
	FOR icounter := 0 TO (ipublishers-1) DO		
		publishers[icounter].Init(inputMQTT_IN_OUT:= ADR(MQTT_IN_OUT));
	END_FOR 
	
	(* INIT MQTT SUBSCRIBE STUFF *)
	subscriber_FB_OUTPUT_SWITCH_MQTT.SetMqttInOut(MQTT_IN_OUT:= ADR(MQTT_IN_OUT));	
	subscriber_FB_OUTPUT_COVER_MQTT.SetMqttInOut(MQTT_IN_OUT:= ADR(MQTT_IN_OUT));

END_IF


                    
END_ACTION

ACTION MQTT_PUBLISH:
                      (* allow the rising edge detector to detect a connect/reconnect to the broker, used for  birth message *)
MQTTConnectTrigger(CLK := MQTTInfo.MQTT_CONNECTED);

(* allow the pulse generator to generate a pulse, used for birth message hartbeat *)
MQTTBirthHartbeat(ENQ:=TRUE, PTH:=T#0S, PTL:=MQTTBirthHartbeatTime);

(* Check if this is a new connection due to startup or connection issues *)
IF initMqtt AND (MQTTConnectTrigger.Q OR MQTTBirthHartbeat.Q) THEN
	MQTTPublishBirth := TRUE;
END_IF

(* On connect or reconnect publish a birth message using the dedicated birth publisher *)
IF MQTTPublishBirth THEN
	MQTTBirthPublisher.PublishMessage(MqttMessage := MQTTBirthMessage);
	MQTTPublishBirth:=FALSE;
END_IF


(* Check if Mqtt is initialized AND if there are elements on the queue to process AND if a MQTTbirthmessage has been published successfully *)
IF initMqtt AND NOT(MqttVariables.fbMqttPublishQueue.EMPTY) AND MQTTPublishBirth = FALSE AND MQTTBirthPublisher.SendDone THEN	
	(* Loop through all free publishers untill there are no more elements in the queue or no more free publishers *)
	FOR i:=0 TO (ipublishers-1) DO			
		(* use the publishers that are free  *)
		IF publishers[i].SendDone AND NOT(MqttVariables.fbMqttPublishQueue.EMPTY) THEN	
			(* Pass message from the queue to a publisher *)
			publishers[i].PublishMessage(MqttMessage:= MqttVariables.fbMqttPublishQueue.GetMessage());
		ELSIF MqttVariables.fbMqttPublishQueue.EMPTY THEN
			(* Queue is empty, jump out of the for loop	*)
			EXIT;	
		END_IF
	END_FOR
END_IF


(* If MQTT is initialized, let the MqttPublishWorkers do their work *)
IF initMqtt THEN
	MQTTClient(
		MQTT_IN_OUT:= MQTT_IN_OUT, 
		ENABLE:= TRUE, 
		URL:= broker, 
		TIMEOUT:= T#1S, 
		TLS:= FALSE);		
		
	MQTTBirthPublisher();
	
	FOR i := 0 TO (ipublishers-1) DO
  		publishers[i]();
	END_FOR

END_IF

                    
END_ACTION

ACTION MQTT_SUBSCRIBE:
                      (* If MQTT is initialized, let the subscriber(s) do its work *)
IF initMqtt THEN
	MQTTClient(
		MQTT_IN_OUT:= MQTT_IN_OUT, 
		ENABLE:= TRUE, 
		URL:= broker, 
		TIMEOUT:= T#1S, 
		TLS:= FALSE);

	subscriber_FB_OUTPUT_SWITCH_MQTT(
		Subscribe:= TRUE, 
		Topic:= ADR('WAGO-PFC200/In/DigitalOutputs/+'), 
		QoSSubscribe:= SD_MQTT.QoS.ExactlyOnce, 
		ExpectingString:= TRUE, 
		Callback:= MqttVariables.collector_FB_OUTPUT_SWITCH_MQTT,
	);
	
	subscriber_FB_OUTPUT_COVER_MQTT(
		Subscribe:= TRUE, 
		Topic:= ADR('WAGO-PFC200/In/Covers/+'), 
		QoSSubscribe:= SD_MQTT.QoS.ExactlyOnce, 
		ExpectingString:= TRUE, 
		Callback:= MqttVariables.collector_FB_OUTPUT_COVER_MQTT,
	);
END_IF

                    
END_ACTION
END_PROGRAM

{attribute 'reflection'}
FUNCTION_BLOCK FB_INPUT_BINARYSENSOR_MQTT
  VAR_INPUT
    BS : BOOL;
  END_VAR
  VAR_OUTPUT
    Q : BOOL;  (* Follows the input but debounced *)
    EVENT : BOOL;  (* Event outputs only high for on clock cycle *)
    EVENT_R : BOOL;
    EVENT_F : BOOL;
  END_VAR
  VAR
    {attribute 'instance-path'}
    {attribute 'noinit'}
    InstanceName : STRING;  (* object's full instance name *)
    InitMqttDone : BOOL;
    MqttPublishTopicPrefix : POINTER TO STRING;
    MqttPublishTopicSuffix : STRING(15);
    pMqttPublishQueue : POINTER TO FB_MqttPublishQueue;
    FB_DEBOUNCE : OSCAT_BUILDING.DEBOUNCE;  (* to debounce the physical input *)
    FB_R_TRIG : Standard.R_TRIG;  (* to detect a rising edge on the debounced signal *)
    FB_F_TRIG : Standard.F_TRIG;  (* to detect a falling edge on the debounced signal *)
  END_VAR

                  FB_DEBOUNCE(IN := BS,	
	TD := T#50MS, (* 2x cyle + 10ms *)
	PM := FALSE,
	Q=>Q);

FB_R_TRIG(CLK := FB_DEBOUNCE.Q);
FB_F_TRIG(CLK := FB_DEBOUNCE.Q);

EVENT := FB_R_TRIG.Q OR FB_F_TRIG.Q;
EVENT_R := FB_R_TRIG.Q;
EVENT_F := FB_F_TRIG.Q;

IF FB_R_TRIG.Q AND InitMqttDone THEN
	pMqttPublishQueue^.AddMessage(
		Payload := 'ON',
		Topic := CONCAT(MqttPublishTopicPrefix^, MqttPublishTopicSuffix),
		Qos := SD_MQTT.QoS.ExactlyOnce,
		MqttRetain := TRUE
	);
END_IF

IF FB_F_TRIG.Q AND InitMqttDone THEN
	pMqttPublishQueue^.AddMessage(
		Payload := 'OFF',
		Topic := CONCAT(MqttPublishTopicPrefix^, MqttPublishTopicSuffix),
		Qos := SD_MQTT.QoS.ExactlyOnce,
		MqttRetain := TRUE
	);
END_IF
                

METHOD InitMqtt
  VAR_INPUT
    MQTTPublishPrefix : POINTER TO STRING;
    pMqttPublishQueue : POINTER TO FB_MqttPublishQueue;
  END_VAR
  VAR
    InstanceNamePt : POINTER TO STRING;
  END_VAR
                        THIS^.pMqttPublishQueue := pMqttPublishQueue;
THIS^.MqttPublishTopicPrefix := MQTTPublishPrefix;

InstanceNamePt := CommonTypesAndFunctions.FindLastDot(ADR(THIS^.InstanceName)) + 1;
THIS^.MqttPublishTopicSuffix := InstanceNamePt^;

InitMqttDone := TRUE;
                      
END_METHOD
END_FUNCTION_BLOCK

{attribute 'reflection'}
FUNCTION_BLOCK FB_INPUT_PUSHBUTTON_DIMMER_MQTT
  VAR_INPUT
    PB : BOOL;
    SET : BOOL;
    VAL : BYTE;
    RST : BOOL;
  END_VAR
  VAR_OUTPUT
    DIM : BYTE;
    DBL : BOOL;
    Q : BOOL;
    SINGLE : BOOL;
    DOUBLE : BOOL;
    LONG : BOOL;
    P_LONG : BOOL;
  END_VAR
  VAR
    {attribute 'instance-path'}
    {attribute 'noinit'}
    InstanceName : STRING;  (* object's full instance name *)
    InitMqttDone : BOOL;
    MqttPublishTopicPrefix : POINTER TO STRING;
    MqttPublishTopicSuffix : STRING(15);
    pMqttPublishQueue : POINTER TO FB_MqttPublishQueue;
    FB_DIMMER : OSCAT_BUILDING.DIMM_I;
    OutputDimmer : BOOL;
    Qos_Dimm : SD_MQTT.QoS;
    Delta_Dimm : INT;
    FB_DETECTPUSH : OSCAT_BUILDING.CLICK_MODE;
    P_LONG_R_TRIG : Standard.R_TRIG;
    P_LONG_F_TRIG : Standard.F_TRIG;
    PreviousDim : BYTE;  (* Vars to detect statechanges on outputs *)
    PreviousQ : BOOL;
    PreviousDBL : BOOL;
    T_Debounce : TIME := TIME#10ms;  (* Default values for dimmer, can be overwritten by method call *)
    T_Reconfig : TIME := TIME#10s0ms;
    T_On_Max : TIME := TIME#0ms;
    T_Dimm_Start : TIME := TIME#400ms;
    T_Dimm : TIME := TIME#3s0ms;
    Min_On : BYTE := 50;
    Max_On : BYTE := 255;
    Soft_Dimm : BOOL := TRUE;
    Dbl_Toggle : BOOL := FALSE;
    Rst_Out : BOOL := FALSE;
    T_Long : TIME := TIME#400ms;  (* Default value for click mode, can be overwritten by method call *)
  END_VAR

                  FB_DIMMER(
	IN:= PB,
	SET:= SET,
	VAL:= VAL,
	RST:= RST,
	OUT:= DIM,
	T_DEBOUNCE:= T_Debounce,
	T_RECONFIG:= T_Reconfig,
	T_ON_MAX:= T_On_Max,
	T_DIMM_START:= T_Dimm_Start,
	T_DIMM:= T_Dimm,
	MIN_ON:= Min_On,
	MAX_ON:= Max_On,
	SOFT_DIMM:= Soft_Dimm,
	DBL_TOGGLE:= Dbl_Toggle,
	RST_OUT:= Rst_Out,
	Q=> Q,
	DBL=> DBL);
	
FB_DETECTPUSH(
	IN:= PB, 	
	SINGLE=> SINGLE, 
	DOUBLE=> DOUBLE, 
	TP_LONG=> LONG, 
	T_LONG:= T_long);
	
P_LONG_R_TRIG(CLK:=FB_DETECTPUSH.LONG);
P_LONG_F_TRIG(CLK:=FB_DETECTPUSH.LONG);
	
IF (ABS(BYTE_TO_INT(PreviousDim) - BYTE_TO_INT(DIM)) >= Delta_Dimm OR PB = FALSE) AND DIM <> PreviousDim AND InitMqttDone AND OutputDimmer THEN
	PreviousDim:=DIM;
	pMqttPublishQueue^.AddMessage(		
		Payload := BYTE_TO_STRING(DIM),
		Topic := CONCAT(CONCAT(MqttPublishTopicPrefix^, MqttPublishTopicSuffix), '/DIM'),
		Qos := SD_MQTT.QoS.ExactlyOnce,
		MqttRetain := FALSE
	);
END_IF

IF FB_DIMMER.Q <> PreviousQ AND InitMqttDone THEN
	PreviousQ:=FB_DIMMER.Q;
	pMqttPublishQueue^.AddMessage(
		Payload := BOOL_TO_STRING(FB_DIMMER.Q),
		Topic := CONCAT(CONCAT(MqttPublishTopicPrefix^, MqttPublishTopicSuffix), '/Q'),
		Qos := Qos_Dimm,
		MqttRetain := TRUE
	);
END_IF

IF FB_DIMMER.DBL <> PreviousDBL AND InitMqttDone THEN
	PreviousDBL:=FB_DIMMER.DBL;
	pMqttPublishQueue^.AddMessage(
		Payload := BOOL_TO_STRING(FB_DIMMER.DBL),
		Topic := CONCAT(CONCAT(MqttPublishTopicPrefix^, MqttPublishTopicSuffix), '/DBL'),
		Qos := SD_MQTT.QoS.ExactlyOnce,
		MqttRetain := TRUE
	);
END_IF

IF FB_DETECTPUSH.SINGLE AND InitMqttDone THEN
	pMqttPublishQueue^.AddMessage(
		Payload := 'SINGLE',
		Topic := CONCAT(MqttPublishTopicPrefix^, MqttPublishTopicSuffix),
		Qos := SD_MQTT.QoS.ExactlyOnce,
		MqttRetain := FALSE
	);
END_IF

IF FB_DETECTPUSH.DOUBLE AND InitMqttDone THEN
	pMqttPublishQueue^.AddMessage(
		Payload := 'DOUBLE',
		Topic := CONCAT(MqttPublishTopicPrefix^, MqttPublishTopicSuffix),
		Qos := SD_MQTT.QoS.ExactlyOnce,
		MqttRetain := FALSE
	);
END_IF

IF FB_DETECTPUSH.TP_LONG AND InitMqttDone THEN
	pMqttPublishQueue^.AddMessage(
		Payload := 'LONG',
		Topic := CONCAT(MqttPublishTopicPrefix^, MqttPublishTopicSuffix),
		Qos := SD_MQTT.QoS.ExactlyOnce,
		MqttRetain := FALSE
	);
END_IF

IF (P_LONG_R_TRIG.Q OR P_LONG_F_TRIG.Q) AND InitMqttDone THEN
	pMqttPublishQueue^.AddMessage(
		Payload := BOOL_TO_STRING(FB_DETECTPUSH.LONG),
		Topic := CONCAT(CONCAT(MqttPublishTopicPrefix^, MqttPublishTopicSuffix),'/P_LONG'),
		Qos := SD_MQTT.QoS.ExactlyOnce,
		MqttRetain := TRUE
	);
END_IF
                

METHOD InitMqtt
  VAR_INPUT
    MQTTPublishPrefix : POINTER TO STRING;
    pMqttPublishQueue : POINTER TO FB_MqttPublishQueue;
    OutputDimmer : BOOL;
    Qos_Dimm : SD_MQTT.QoS;
    Delta_Dimm : INT;
  END_VAR
  VAR
    InstanceNamePt : POINTER TO STRING;
  END_VAR
                        THIS^.pMqttPublishQueue := pMqttPublishQueue;
THIS^.MqttPublishTopicPrefix := MQTTPublishPrefix;

InstanceNamePt := CommonTypesAndFunctions.FindLastDot(ADR(THIS^.InstanceName)) + 1;
THIS^.MqttPublishTopicSuffix := InstanceNamePt^;

THIS^.OutputDimmer:=OutputDimmer;
THIS^.Qos_Dimm:=Qos_Dimm;
THIS^.Delta_Dimm:=Delta_Dimm;

InitMqttDone := TRUE;
                      
END_METHOD

METHOD ConfigureFunctionBlock
  VAR_INPUT
    T_Debounce : TIME;  (* Default values for dimmer, can be overwritten by method call *)
    T_Reconfig : TIME;
    T_On_Max : TIME;
    T_Dimm_Start : TIME;
    T_Dimm : TIME;
    Min_On : BYTE;
    Max_On : BYTE;
    Soft_Dimm : BOOL;
    Dbl_Toggle : BOOL;
    Rst_Out : BOOL;
    T_Long : TIME;  (* Default value for click mode, can be overwritten by method call *)
  END_VAR
                        THIS^.T_Debounce:=T_Debounce;
THIS^.T_Reconfig:=T_Reconfig;
THIS^.T_On_Max:=T_On_Max;
THIS^.T_Dimm_Start:=T_Dimm_Start;
THIS^.T_Dimm:=T_Dimm;
THIS^.Min_On:=Min_On;
THIS^.Max_On:=Max_On;

THIS^.T_Long:=T_Long;
                      
END_METHOD
END_FUNCTION_BLOCK

FUNCTION_BLOCK _RMP_B
  VAR_INPUT
    DIR : BOOL;  (* true = up *)
    E : BOOL := TRUE;
    TR : TIME;
  END_VAR
  VAR_IN_OUT
    RMP : BYTE;
  END_VAR
  VAR
    tx : TIME;
    tl : TIME;
    tn : TIME;
    init : BOOL;
    last_dir : BOOL;
    start : BYTE;
  END_VAR

                  (* read system timer *)
tx := DWORD_TO_TIME(OSCAT_BASIC.T_PLC_MS());

IF E AND init AND (dir = last_dir) AND (RMP <> SEL(DIR, 0, 255)) AND TR = tn THEN
	RMP := OSCAT_BASIC.FRMP_B(start, DIR, tx - tl, TR);
ELSE
	init := TRUE;
	tl := tx;
	tn := tr;
	start := RMP;
END_IF;
last_dir := dir;



(* revison history
hm	22. oct. 2008	rev 1.0
	original version

hm	20. nov. 2008	rev 1.1
	set default for E to be TRUE
	added init

hm	19. nov. 2011	rev 1.2
	new code
*)
                

METHOD SetRMP
  VAR_INPUT
    RMP : BYTE;
  END_VAR
                        (*THIS^.RMP:=RMP;*)
THIS^.Start:=RMP;
                      
END_METHOD
END_FUNCTION_BLOCK

FUNCTION_BLOCK RMP_B
  VAR_INPUT
    SET : BOOL;
    PT : TIME;
    E : BOOL := TRUE;
    UP : BOOL := TRUE;
    RST : BOOL;
  END_VAR
  VAR_OUTPUT
    OUT : BYTE;
    BUSY : BOOL;
    HIGH : BOOL;
    LOW : BOOL;
  END_VAR
  VAR
    rmp : _RMP_B;
  END_VAR

                  (* generate ramp *)
rmp(dir := UP, E := E, TR := PT, rmp := out);

(* set or reset operation *)
IF RST THEN
	out := 0;
ELSIF SET THEN
	out := 255;
END_IF;

(* checks for outputs stable and reset or set busy flag *)
low := out = 0;
high := out = 255;
busy := NOT (low OR high) AND E;


(* revision history

hm 5.10.2006	rev 1.1
	added busy output
hm 17.1.2007	rev 1.2
	renamed input ud to up for better usability
	deleted unused variable step

hm	17.9.2007		rev 1.3
	replaced time() with t_plc_ms() for compatibility reasons

hm	28. sep 2007	rev 1.4
	added outputs on and off
	busy is now disabled while en is false
	new coding for higher accuracy and performance

hm	5. oct 2007	rev 1.5
	added statements to allow for PT to be t#0s output jumps to max or min immediately

hm	25. dec 2007	rev 1.6
	improved code for better performance

hm	16. oct. 2008	rev 1.7
	improved code for better performance

hm	18. oct. 2008	rev 1.8
	added type conversion to avoid warnings
	changed input en to e for compatibility reasons

hm	23. oct. 2008	REV 	2.0
	new code using _RMP_B

*)
                

METHOD SetRMP
  VAR_INPUT
    RMP : BYTE;
  END_VAR
                        THIS^.OUT:=RMP;
THIS^.rmp.SetRMP(RMP);
                      
END_METHOD
END_FUNCTION_BLOCK

FUNCTION_BLOCK BLIND_ACTUATOR
  VAR_INPUT
    UP : BOOL;
    DN : BOOL;
    S_IN : BYTE;
    T_UD : TIME := TIME#10s0ms;
    T_ANGLE : TIME := TIME#3s0ms;
    {attribute 'input_constant'}
    T_LOCKOUT : TIME := TIME#100ms;
  END_VAR
  VAR_OUTPUT
    POS : BYTE;
    ANG : BYTE;
    QU : BOOL;
    QD : BOOL;
    STATUS : BYTE;
  END_VAR
  VAR
    position : RMP_B;
    angle : RMP_B;
    lock : OSCAT_BASIC.INTERLOCK;
  END_VAR

                  (* make sure only one motor is active at a given time *)
lock(i1 := UP, I2 := DN, TL := T_lockout);

(* ramp up or down to simulate the angle position of the blind slats *)
angle(e := lock.Q1 OR lock.Q2, UP := lock.Q1, PT := T_Angle);
position(e := lock.Q1 AND angle.high OR lock.Q2 AND angle.low, up := lock.Q1, PT := T_UD);

(* set the outputs *)
pos := position.Out;
ang := angle.Out;

(* set the outputs *)
QU := lock.Q1;
QD := lock.Q2;

(* set the status output *)
IF UP AND DN THEN
	 status := 1;			(* error up and down together are not allowed *)
ELSIF UP THEN
	status := 121;
ELSIF DN THEN
	status := 122;
ELSE
	status := S_IN;
END_IF;


(* revision history
hm	29. sep 2007	rev 1.0
	original release

hm	6. oct 2007	rev 1.1
	rearanged outputs

hm	18. oct. 2008	rev 1.2
	changed calls for rmp_B because of change in RMP_B

hm	27. jul. 2009	rev 1.3
	changes status to be 12X

ae	08. mar. 2010 rev 1.4	
	at aPosition

*)
                

METHOD SetPOS
  VAR_INPUT
    POS : BYTE;
  END_VAR
                        THIS^.POS:=POS;
THIS^.position.SetRMP(POS);
                      
END_METHOD
END_FUNCTION_BLOCK

{attribute 'reflection'}
FUNCTION_BLOCK FB_OUTPUT_COVER_MQTT IMPLEMENTS SD_MQTT.MQTT_SUBSCRIBE_CALLBACK
  VAR_INPUT
    UP : BOOL;
    DN : BOOL;
    PI : BYTE;
    PRIO_LOCK : BOOL;
    PRIO_UP : BOOL;
    PRIO_DN : BOOL;
    {attribute 'input_constant'}
    SENS : BYTE := 1;
    {attribute 'input_constant'}
    T_LOCKOUT : TIME := TIME#1s0ms;
    {attribute 'input_constant'}
    T_UD : TIME := TIME#10s0ms;
  END_VAR
  VAR_OUTPUT
    POS : BYTE;
    MU : BOOL;
    MD : BOOL;
  END_VAR
  VAR
    {attribute 'instance-path'}
    {attribute 'noinit'}
    InstanceName : STRING;  (* object's full instance name *)
    Startup : BOOL := TRUE;
    InitMqttDone : BOOL;
    MqttPublishTopicPrefix : POINTER TO STRING;
    MqttPublishTopicSuffix : STRING(15);
    MQTTSubscribeTopic : STRING(50);
    pMqttPublishQueue : POINTER TO FB_MqttPublishQueue;
    FB_ACT : BLIND_ACTUATOR;
    delta : BYTE;
    internal_UP : BOOL;
    internal_DN : BOOL;
    Qos_POS : SD_MQTT.QoS;
    Delta_POS : INT;
    Cover_State : COVER_STATES;
    Cover_State_Timer : TOF;
    MqttRequestAuto : BOOL;
    MqttRequestStop : BOOL;
    MqttRequestCalibrateUp : BOOL;
    MqttRequestCalibrateDn : BOOL;
  END_VAR
  VAR PERSISTENT
    PreviousPos : BYTE;  (* To retain position through powercycles *)
  END_VAR

                  IF Startup THEN
	POS:=PreviousPos;
	FB_ACT.SetPOS(PreviousPos);
END_IF

Cover_State_Timer(PT:=2 * T_UD);
Cover_State_Timer.IN:=FALSE;

CASE Cover_State OF
	COVER_STATES.Idle:
		internal_UP:=FALSE;
		internal_DN:=FALSE;
		//Calculate the next state
		Cover_State := CALC_COVER_STATE(UP:=UP,DN:=DN,PRIO_LOCK:=PRIO_LOCK,PRIO_UP:=PRIO_UP,PRIO_DN:=PRIO_DN,PI:=PI,POS:=POS,MqttRequestAuto:=ADR(MqttRequestAuto),MqttRequestStop:=ADR(MqttRequestStop),MqttRequestCalibrateUp:=ADR(MqttRequestCalibrateUp),MqttRequestCalibrateDn:=ADR(MqttRequestCalibrateDn),CurrentState:=Cover_State,StateTimer:=ADR(Cover_State_Timer));
	COVER_STATES.Prio_up:
		// Only power an engine for maximum twice T_UD
		IF Cover_State_Timer.Q THEN
			internal_UP:=TRUE;
			internal_DN:=FALSE;
		ELSE
			internal_UP:=FALSE;
			internal_DN:=FALSE;
		END_IF
		//Calculate the next state
		Cover_State := CALC_COVER_STATE(UP:=UP,DN:=DN,PRIO_LOCK:=PRIO_LOCK,PRIO_UP:=PRIO_UP,PRIO_DN:=PRIO_DN,PI:=PI,POS:=POS,MqttRequestAuto:=ADR(MqttRequestAuto),MqttRequestStop:=ADR(MqttRequestStop),MqttRequestCalibrateUp:=ADR(MqttRequestCalibrateUp),MqttRequestCalibrateDn:=ADR(MqttRequestCalibrateDn),CurrentState:=Cover_State,StateTimer:=ADR(Cover_State_Timer));
	COVER_STATES.Prio_dn:
		// Only power an engine for maximum twice T_UD
		IF Cover_State_Timer.Q THEN
			internal_UP:=FALSE;
			internal_DN:=TRUE;
		ELSE
			internal_UP:=FALSE;
			internal_DN:=FALSE;
		END_IF
		//Calculate the next state
		Cover_State := CALC_COVER_STATE(UP:=UP,DN:=DN,PRIO_LOCK:=PRIO_LOCK,PRIO_UP:=PRIO_UP,PRIO_DN:=PRIO_DN,PI:=PI,POS:=POS,MqttRequestAuto:=ADR(MqttRequestAuto),MqttRequestStop:=ADR(MqttRequestStop),MqttRequestCalibrateUp:=ADR(MqttRequestCalibrateUp),MqttRequestCalibrateDn:=ADR(MqttRequestCalibrateDn),CurrentState:=Cover_State,StateTimer:=ADR(Cover_State_Timer));
	COVER_STATES.Auto:
		internal_UP:=TRUE;
		internal_DN:=TRUE;
		//Calculate the next state
		Cover_State := CALC_COVER_STATE(UP:=UP,DN:=DN,PRIO_LOCK:=PRIO_LOCK,PRIO_UP:=PRIO_UP,PRIO_DN:=PRIO_DN,PI:=PI,POS:=POS,MqttRequestAuto:=ADR(MqttRequestAuto),MqttRequestStop:=ADR(MqttRequestStop),MqttRequestCalibrateUp:=ADR(MqttRequestCalibrateUp),MqttRequestCalibrateDn:=ADR(MqttRequestCalibrateDn),CurrentState:=Cover_State,StateTimer:=ADR(Cover_State_Timer));
	COVER_STATES.Manual:
		internal_UP:=UP;
		internal_DN:=DN;
		//Calculate the next state
		Cover_State := CALC_COVER_STATE(UP:=UP,DN:=DN,PRIO_LOCK:=PRIO_LOCK,PRIO_UP:=PRIO_UP,PRIO_DN:=PRIO_DN,PI:=PI,POS:=POS,MqttRequestAuto:=ADR(MqttRequestAuto),MqttRequestStop:=ADR(MqttRequestStop),MqttRequestCalibrateUp:=ADR(MqttRequestCalibrateUp),MqttRequestCalibrateDn:=ADR(MqttRequestCalibrateDn),CurrentState:=Cover_State,StateTimer:=ADR(Cover_State_Timer));
	COVER_STATES.Calibrate_up:
		// Only power an engine for maximum twice T_UD
		IF Cover_State_Timer.Q THEN
			internal_UP:=FALSE;
			internal_DN:=TRUE;
		ELSE
			internal_UP:=FALSE;
			internal_DN:=FALSE;
			//Finish the request
			MqttRequestCalibrateUp:=FALSE;
		END_IF
		//Calculate the next state
		Cover_State := CALC_COVER_STATE(UP:=UP,DN:=DN,PRIO_LOCK:=PRIO_LOCK,PRIO_UP:=PRIO_UP,PRIO_DN:=PRIO_DN,PI:=PI,POS:=POS,MqttRequestAuto:=ADR(MqttRequestAuto),MqttRequestStop:=ADR(MqttRequestStop),MqttRequestCalibrateUp:=ADR(MqttRequestCalibrateUp),MqttRequestCalibrateDn:=ADR(MqttRequestCalibrateDn),CurrentState:=Cover_State,StateTimer:=ADR(Cover_State_Timer));
	COVER_STATES.Calibrate_dn:
		// Only power an engine for maximum twice T_UD
		IF Cover_State_Timer.Q THEN
			internal_UP:=FALSE;
			internal_DN:=TRUE;
		ELSE
			internal_UP:=FALSE;
			internal_DN:=FALSE;
			//Finish the request
			MqttRequestCalibrateDn:=FALSE;
		END_IF
		//Calculate the next state
		Cover_State := CALC_COVER_STATE(UP:=UP,DN:=DN,PRIO_LOCK:=PRIO_LOCK,PRIO_UP:=PRIO_UP,PRIO_DN:=PRIO_DN,PI:=PI,POS:=POS,MqttRequestAuto:=ADR(MqttRequestAuto),MqttRequestStop:=ADR(MqttRequestStop),MqttRequestCalibrateUp:=ADR(MqttRequestCalibrateUp),MqttRequestCalibrateDn:=ADR(MqttRequestCalibrateDn),CurrentState:=Cover_State,StateTimer:=ADR(Cover_State_Timer));
	ELSE
		Cover_State:=COVER_STATES.Idle;
END_CASE

(* Check Position*)
FB_ACT(T_UD:=T_UD, T_ANGLE:=T#0S, T_lockout := T_Lockout);

IF internal_UP AND internal_DN THEN
	(* automatic modus detected *)
	(* first find correct position *)
	IF BYTE_TO_INT(FB_ACT.pos) < BYTE_TO_INT(pi) - delta THEN
		FB_ACT.UP := TRUE;
		FB_ACT.DN := FALSE;
		delta := 0;
	ELSIF BYTE_TO_INT(FB_ACT.pos) > BYTE_TO_INT(pi) + delta THEN
		FB_ACT.UP := FALSE;
		FB_ACT.DN := TRUE;
		delta := 0;
	(* correct position reached *)
	ELSE
		FB_ACT.UP := FALSE;
		FB_ACT.DN := FALSE;
		delta := sens;
	END_IF;
ELSE
	FB_ACT.UP := internal_UP;
	FB_ACT.DN := internal_DN;
END_IF;

(* blind control calls blind_actuator *)
FB_ACT(T_UD:=T_UD, T_ANGLE:=T#0S, T_lockout := T_Lockout);
POS := FB_ACT.pos;
MU := FB_ACT.QU;
MD := FB_ACT.QD;

IF (ABS(BYTE_TO_INT(PreviousPos) - BYTE_TO_INT(POS)) >= Delta_POS  OR (MU = FALSE AND MD = FALSE)) AND POS <> PreviousPos OR Startup AND InitMqttDone THEN
	PreviousPos:=POS;
	pMqttPublishQueue^.AddMessage(
		Payload := INT_TO_STRING(REAL_TO_INT(OSCAT_BASIC.SCALE_B(X:=POS, I_LO:=0, I_HI:=255, O_LO:=0, O_HI:=100))),
		Topic := CONCAT(MqttPublishTopicPrefix^, MqttPublishTopicSuffix),
		Qos := Qos_POS,
		MqttRetain := TRUE
	);
	Startup:=FALSE;
END_IF

                

METHOD InitMqtt
  VAR_INPUT
    MQTTPublishPrefix : POINTER TO STRING;
    MQTTSubscribePrefix : POINTER TO STRING;
    pMqttPublishQueue : POINTER TO FB_MqttPublishQueue;
    pMqttCallbackCollector : POINTER TO SD_MQTT.CallbackCollector;
    Qos_POS : SD_MQTT.QoS;
    Delta_POS : INT;
  END_VAR
  VAR
    InstanceNamePt : POINTER TO STRING;
  END_VAR
                        THIS^.pMqttPublishQueue := pMqttPublishQueue;
THIS^.MqttPublishTopicPrefix := MQTTPublishPrefix;

InstanceNamePt := CommonTypesAndFunctions.FindLastDot(ADR(THIS^.InstanceName)) + 1;
THIS^.MqttPublishTopicSuffix := InstanceNamePt^;
THIS^.MQTTSubscribeTopic := CONCAT(MQTTSubscribePrefix^ ,THIS^.MqttPublishTopicSuffix);

// register the FB agains the collector so mqtt events can be received
pMqttCallbackCollector^.put(instance:= THIS^);

THIS^.Qos_POS:=Qos_POS;
THIS^.Delta_POS:=REAL_TO_INT(OSCAT_BASIC.SCALE_B(X:=INT_TO_BYTE(Delta_POS), I_LO:=0, I_HI:=100, O_LO:=0, O_HI:=255));

InitMqttDone := TRUE;
                      
END_METHOD

METHOD PublishReceived : BOOL
  VAR_INPUT
    Data : SD_MQTT.CALLBACK_DATA;  (* Collection of recived Data *)
  END_VAR
                        //first check if Mqtt is initialized, otherwise do nothing
IF NOT(InitMqttDone) THEN
	//mark the interface call from the collector as done
	PublishReceived := TRUE;
//check if the packet is for this FB
ELSIF CommonTypesAndFunctions.StrEquals(str1:= ADR(MQTTSubscribeTopic), str2:= Data.TopicOut) THEN
	//mark the interface call from the collector as done
	PublishReceived := TRUE;
	//now process the data
	IF CommonTypesAndFunctions.StrEquals(str1:= Data.PayloadString, str2:= ADR('STOP')) THEN			
		THIS^.MqttRequestStop:=TRUE;
	ELSIF CommonTypesAndFunctions.StrEquals(str1:= Data.PayloadString, str2:= ADR('OPEN')) THEN
		THIS^.PI:=255;
		THIS^.MqttRequestAuto:=TRUE;
	ELSIF CommonTypesAndFunctions.StrEquals(str1:= Data.PayloadString, str2:= ADR('CLOSE')) THEN		
		THIS^.PI:=0;
		THIS^.MqttRequestAuto:=TRUE;
	ELSIF CommonTypesAndFunctions.StrEquals(str1:= Data.PayloadString, str2:= ADR('CAL_UP')) THEN
		THIS^.MqttRequestCalibrateUp:=TRUE;
	ELSIF CommonTypesAndFunctions.StrEquals(str1:= Data.PayloadString, str2:= ADR('CAL_DN')) THEN
		THIS^.MqttRequestCalibrateDn:=TRUE;
	ELSIF OSCAT_BASIC.IS_NUM(str:= Data.PayloadString^) THEN
		THIS^.PI:=REAL_TO_BYTE(OSCAT_BASIC.SCALE_B(X:=STRING_TO_BYTE(Data.PayloadString^), I_LO:=0, I_HI:=100, O_LO:=0, O_HI:=255));
		THIS^.MqttRequestAuto:=TRUE;
	END_IF

END_IF 
                      
END_METHOD

METHOD ConfigureFunctionBlock : BOOL
  VAR_INPUT
    T_LOCKOUT : TIME;
    T_UD : TIME;
  END_VAR
                        THIS^.T_LOCKOUT:=T_LOCKOUT;
THIS^.T_UD:=T_UD;
                      
END_METHOD
END_FUNCTION_BLOCK

FUNCTION CALC_COVER_STATE : COVER_STATES
  VAR_INPUT
    UP : BOOL;
    DN : BOOL;
    PRIO_LOCK : BOOL;
    PRIO_UP : BOOL;
    PRIO_DN : BOOL;
    PI : BYTE;
    POS : BYTE;
    MqttRequestAuto : POINTER TO BOOL;
    MqttRequestStop : POINTER TO BOOL;
    MqttRequestCalibrateUp : POINTER TO BOOL;
    MqttRequestCalibrateDn : POINTER TO BOOL;
    CurrentState : COVER_STATES;
    StateTimer : POINTER TO TOF;
  END_VAR
  VAR
    NewState : COVER_STATES;
  END_VAR

                  IF PRIO_LOCK THEN
	NewState := COVER_STATES.Idle;
	MqttRequestAuto^ := FALSE;
	MqttRequestStop^ := FALSE;
	MqttRequestCalibrateUp^ := FALSE;
	MqttRequestCalibrateDn^ := FALSE;
ELSIF PRIO_UP THEN
	NewState := COVER_STATES.Prio_up;
	MqttRequestAuto^ := FALSE;
	MqttRequestStop^ := FALSE;
	MqttRequestCalibrateUp^ := FALSE;
	MqttRequestCalibrateDn^ := FALSE;
ELSIF PRIO_DN THEN
	NewState := COVER_STATES.Prio_dn;
	MqttRequestAuto^ := FALSE;
	MqttRequestStop^ := FALSE;
	MqttRequestCalibrateUp^ := FALSE;
	MqttRequestCalibrateDn^ := FALSE;
ELSIF UP OR DN THEN
	NewState := COVER_STATES.Manual;
	MqttRequestAuto^ := FALSE;
	MqttRequestStop^ := FALSE;
	MqttRequestCalibrateUp^ := FALSE;
	MqttRequestCalibrateDn^ := FALSE;
ELSIF MqttRequestStop^ THEN
	NewState := COVER_STATES.Idle;
	MqttRequestAuto^ := FALSE;
	MqttRequestStop^ := FALSE;
	MqttRequestCalibrateUp^ := FALSE;
	MqttRequestCalibrateDn^ := FALSE;
ELSIF MqttRequestAuto^ AND PI <> POS THEN
	NewState := COVER_STATES.Auto;
	MqttRequestStop^ := FALSE;
	MqttRequestCalibrateUp^ := FALSE;
	MqttRequestCalibrateDn^ := FALSE;
ELSIF MqttRequestAuto^ AND PI = POS THEN
	NewState := COVER_STATES.Idle;
	MqttRequestAuto^ := FALSE;
	MqttRequestStop^ := FALSE;
	MqttRequestCalibrateUp^ := FALSE;
	MqttRequestCalibrateDn^ := FALSE;
ELSIF MqttRequestCalibrateUp^ THEN
	NewState := COVER_STATES.Calibrate_up;
	MqttRequestAuto^ := FALSE;
	MqttRequestStop^ := FALSE;
	MqttRequestCalibrateDn^ := FALSE;
ELSIF MqttRequestCalibrateDn^ THEN
	NewState := COVER_STATES.Calibrate_dn;
	MqttRequestAuto^ := FALSE;
	MqttRequestStop^ := FALSE;
	MqttRequestCalibrateDn^ := FALSE;
ELSE
	NewState := COVER_STATES.Idle;
	MqttRequestAuto^ := FALSE;
	MqttRequestStop^ := FALSE;
	MqttRequestCalibrateUp^ := FALSE;
	MqttRequestCalibrateDn^ := FALSE;
END_IF

IF NewState <> CurrentState THEN
	//Reset StateTimer
	StateTimer^.IN:=TRUE;
END_IF

CALC_COVER_STATE := NewState;
                
END_FUNCTION

CONFIGURATION Application
  RESOURCE HomeAutomation ON PLC
    {attribute 'qualified_only'}
    VAR_GLOBAL  (* MqttVariables *)
      fbMqttPublishQueue : FB_MqttPublishQueue;  (* Shared Variables for MQTT publish communication *)
      collector_FB_OUTPUT_SWITCH_MQTT : SD_MQTT.CallbackCollector;  (* Shared Variables for MQTT subscribe communication *)
      collector_FB_OUTPUT_COVER_MQTT : SD_MQTT.CallbackCollector;
    END_VAR
    TASK MainTask(INTERVAL := T#20ms, PRIORITY := 0);
    TASK MqttCommunication(PRIORITY := 1);
    PROGRAM PLC_PRG_MAIN WITH MainTask : PLC_PRG_MAIN;
    PROGRAM PLC_PRG_MQTT WITH MqttCommunication : PLC_PRG_MQTT;
  END_RESOURCE
END_CONFIGURATION
